FUNCTION_BLOCK PAEEMotorStartCtrl EXTENDS PAEEMotorBase
VAR_INPUT
END_VAR
VAR_OUTPUT
END_VAR
VAR
	_ChangeoverDelay : TIME;
	_ReqSpeed : LREAL;
	_StarterState : PANotifyState;
	_StarterStateACK : BOOL;
	_TransitTimeStar : TIME;
END_VAR

{attribute 'monitoring' := 'call'}
//{attribute 'TcRpcEnable'}
PROPERTY PUBLIC ChangeoverDelay : TIME
GET // PUBLIC
ChangeoverDelay := _ChangeoverDelay;
END_GET
SET // PUBLIC
_ChangeoverDelay := ChangeoverDelay;
Root.OnPropertyChangedTime(THIS^, 43, _ChangeoverDelay);
END_SET
END_PROPERTY

METHOD PUBLIC FB_postinit
VAR_INPUT
		root : IACVariobatch;
END_VAR
SUPER^.FB_postinit(root);  
root.OnPropertyChangedTime(THIS^, 42, _TransitTimeStar);
root.OnPropertyChangedTime(THIS^, 43, _ChangeoverDelay);
root.OnPropertyChangedInt(THIS^, 44, _StarterState);
root.OnPropertyChangedLReal(THIS^, 45, _ReqSpeed);
root.OnPropertyChangedBool(THIS^, 46, _StarterStateACK);
END_METHOD

METHOD PUBLIC InvokeSetterBool
VAR_INPUT
	PropertyID : INT;
	PropertyValue : BOOL;
END_VAR
SUPER^.InvokeSetterBool(PropertyID, PropertyValue);
CASE PropertyID OF
	46:
		StarterStateACK := PropertyValue;
END_CASE
END_METHOD

METHOD PUBLIC InvokeSetterEnum
VAR_INPUT
	PropertyID : INT;
	PropertyValue : INT;
END_VAR
SUPER^.InvokeSetterEnum(PropertyID, PropertyValue);
IF PropertyID = 44 THEN
	THIS^.StarterState := PropertyValue;
END_IF
END_METHOD

METHOD PUBLIC InvokeSetterLReal
VAR_INPUT
	PropertyID : INT;
	PropertyValue : LREAL;
END_VAR
SUPER^.InvokeSetterLReal(PropertyID, PropertyValue);
CASE PropertyID OF
	45:
		ReqSpeed := PropertyValue;
END_CASE
END_METHOD

METHOD PUBLIC InvokeSetterTime
VAR_INPUT
	PropertyID : INT;
	PropertyValue : DINT;
END_VAR
SUPER^.InvokeSetterTime(PropertyID, PropertyValue);
CASE PropertyID OF
	42:
		TransitTimeStar := TO_TIME(PropertyValue);
	43:
		ChangeoverDelay := TO_TIME(PropertyValue);
END_CASE
END_METHOD

METHOD PUBLIC IsEnabledAcknowledgeAlarms : BOOL
VAR_INPUT
END_VAR
END_METHOD

METHOD OnInitMemory
VAR_INPUT
		root : IACVariobatch;
END_VAR
RegisterProperty(root, 42, GCL.cSizeTIME); //TransitTimeStar
RegisterProperty(root, 43, GCL.cSizeTIME); //ChangeOverDelay
RegisterProperty(root, 44, GCL.cSizeINT); //StarterState
RegisterProperty(root, 45, GCL.cSizeLREAL); //ReqSpeed
RegisterProperty(root, 46, GCL.cSizeBYTE); //StarterStateACK
SUPER^.OnInitMemory(root);
END_METHOD

METHOD PUBLIC OnSetStarterState
VAR_INPUT
END_VAR
END_METHOD

{attribute 'monitoring' := 'call'}
//{attribute 'TcRpcEnable'}
PROPERTY PUBLIC ReqSpeed : LREAL
GET // PUBLIC
ReqSpeed := _ReqSpeed;
END_GET
SET // PUBLIC
_ReqSpeed:=ReqSpeed;
Root.OnPropertyChangedLReal(THIS^, 45, _ReqSpeed);
END_SET
END_PROPERTY

{attribute 'monitoring' := 'call'}
//{attribute 'TcRpcEnable'}
PROPERTY PUBLIC StarterState : PANotifyState
GET // PUBLIC
StarterState := _StarterState;
END_GET
SET // PUBLIC
_StarterState := StarterState;
Root.OnPropertyChangedInt(THIS^, 44, _StarterState);
END_SET
END_PROPERTY

METHOD StarterState_PropertyChanged
VAR_INPUT
END_VAR
END_METHOD

{attribute 'monitoring' := 'call'}
//{attribute 'TcRpcEnable'}
PROPERTY PUBLIC StarterStateACK : BOOL
GET // PUBLIC
StarterStateACK := _StarterStateACK;
END_GET
SET // PUBLIC
_StarterStateACK := StarterStateACK;
Root.OnPropertyChangedBool(THIS^, 46, _StarterStateACK);
END_SET
END_PROPERTY

{attribute 'monitoring' := 'call'}
//{attribute 'TcRpcEnable'}
PROPERTY PUBLIC TransitTimeStar : TIME
GET // PUBLIC
TransitTimeStar := _TransitTimeStar;
END_GET
SET // PUBLIC
_TransitTimeStar := TransitTimeStar;
Root.OnPropertyChangedTime(THIS^, 42, _TransitTimeStar);
END_SET
END_PROPERTY

END_FUNCTION_BLOCK

(* stored: Version 1.1.0.1, ProductVersion 3.1.4024.6
   POU PAEEMotorStartCtrl: Id {36a3067f-bdc9-4d55-a069-de2cd453ef7d}, SpecialFunc None
   Property ChangeoverDelay: Id {0f162ea0-a305-4333-987b-a4039512b76b}
   Get Get: Id {0e35e9bb-1b63-4c5c-8624-79cff4b9f7aa}
   Set Set: Id {f30a59ec-bea3-452a-9647-103ce9557f3e}
   Method FB_postinit: Id {e7439814-43ce-4545-8494-038b96f232ad}
   Method InvokeSetterBool: Id {db6d87f6-9c73-4447-b18a-e7e53c09c77c}
   Method InvokeSetterEnum: Id {be33fc26-b5fa-48bb-8628-fba1a40445c2}
   Method InvokeSetterLReal: Id {c91a4caf-392e-4e9f-8783-090d150ba2a0}
   Method InvokeSetterTime: Id {28a891a1-0cbe-4fa0-84bd-4f806f189a4e}
   Method IsEnabledAcknowledgeAlarms: Id {4c6a12c2-1437-4265-9e05-315281e75900}
   Method OnInitMemory: Id {0d534acf-e779-4e66-a9ab-638e6d7897c9}
   Method OnSetStarterState: Id {8bf5d9cd-e5e3-4b80-b25f-b05f58375a9a}
   Property ReqSpeed: Id {f076b022-70df-420a-b4fc-d66ebacdc8ca}
   Get Get: Id {6937a165-2f9e-4a28-a920-439e39974d39}
   Set Set: Id {11f960eb-678a-4146-92ae-841ae8392a51}
   Property StarterState: Id {b699f06a-61c3-4760-ab24-d86619336bd1}
   Get Get: Id {721f7052-457f-4595-be2c-289ad2346ebf}
   Set Set: Id {fe5e2b75-33c4-49e3-96d7-e3e931fd1106}
   Method StarterState_PropertyChanged: Id {4e4a7675-54e8-43e8-adf3-b54839e077c3}
   Property StarterStateACK: Id {f892bbc7-bf30-46b7-a359-211675b7061c}
   Get Get: Id {1d8583c6-1aad-4f03-8fa1-641b7a591c44}
   Set Set: Id {0bbc8a14-4275-4bd1-bfdf-0191ce5381df}
   Property TransitTimeStar: Id {fded1e13-4123-4d1d-adde-5706a948c0e1}
   Get Get: Id {c43b3e43-e07b-4ac0-9f46-0ce1eaccf658}
   Set Set: Id {2bd14041-fa28-45cf-8546-e1aaaa5fe612} *)
